TYPE st_Device :
STRUCT
	SystemUptime	:	UDINT;	
	Temperature		:	REAL;
	RouterSerial	:	STRING(32);
END_STRUCT
END_TYPE

(* stored: Version 1.1.0.1, ProductVersion 3.1.4024.12
   DUT st_Device: Id {352b9ebc-ec38-4c5d-8e18-14d0766fff60} *)
